// TIA Portal V20 export
FUNCTION "Services" : Void   // FC25, FBD
TITLE = Service
{ S7_Optimized_Access := 'TRUE' }
AUTHOR : Siemens AG
FAMILY : ServiceControl
VERSION : 1.0
// stored: SetENOAutomatically false
   VAR_TEMP
      ProcedureDone : Bool;
      UnholdingDone : Bool;
      StartingState : Bool;
      CompletingState : Bool;
      PausingState : Bool;
      HoldingState : Bool;
      AbortingState : Bool;
      StoppingState : Bool;
   END_VAR
   VAR_TEMP   // added for the SCL form of the ladder/FBD networks
      _w1 : Bool;
      _w2 : Bool;
      _w3 : Bool;
   END_VAR
BEGIN

REGION Network 1: Parameters and values
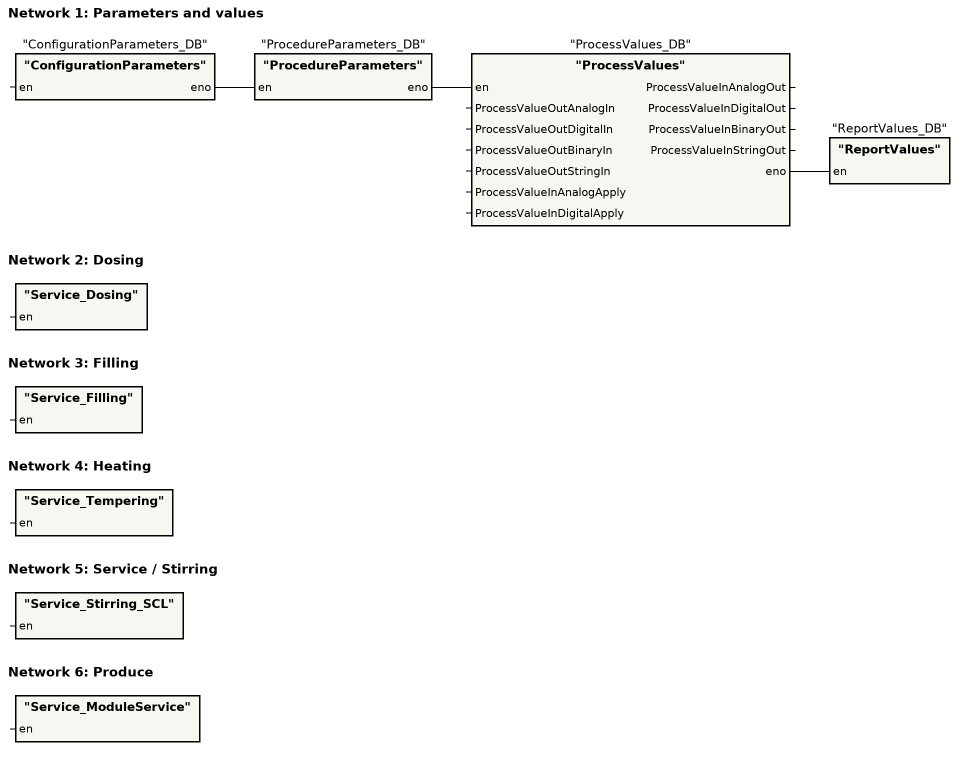
   "ConfigurationParameters_DB"(ENO => #_w1);   // "ConfigurationParameters"
   "ProcedureParameters_DB"(EN := #_w1, ENO => #_w2);   // "ProcedureParameters"
   "ProcessValues_DB"(EN := #_w2, ENO => #_w3);   // "ProcessValues"
   IF #_w3 THEN
       "ReportValues_DB"();   // "ReportValues"
   END_IF;
END_REGION

REGION Network 2: Dosing
   "Service_Dosing"();
END_REGION

REGION Network 3: Filling
   "Service_Filling"();
END_REGION

REGION Network 4: Heating
   "Service_Tempering"();
END_REGION

REGION Network 5: Service / Stirring
   "Service_Stirring_SCL"();
END_REGION

REGION Network 6: Produce
   "Service_ModuleService"();
END_REGION
END_FUNCTION
